// TIA Portal V20 export
// export: Created 2026-08-08T00:00:00.0000000Z, ExportSetting WithDefaults, DisplayName Totally Integrated Automation Portal, DisplayVersion V20, DisplayName TIA Portal Openness, DisplayVersion V20, DisplayName TIA Portal Version Control Interface, DisplayVersion V20, DisplayName STEP 7 Professional, DisplayVersion V20, DisplayName STEP 7 Safety, DisplayVersion V20, DisplayName WinCC Basic/Comfort/Advanced, DisplayVersion V20, DisplayName WinCC Professional, DisplayVersion V20, DisplayName WinCC Unified, DisplayVersion V20
DATA_BLOCK "Valve_Channels_DB"   // DB
{ S7_Optimized_Access := 'TRUE' }
VERSION : 0.1
// Per-valve physical channel assignment table (1..88). All zero until the confirmed valve list / channel schedule is filled in - the mapper and everything downstream treats a zero channel as "use symbolic simulation, no real I/O assigned yet" so this DB is safe to exist unfilled.
// stored: AutoNumber true, IsOnlyStoredInLoadMemory false, IsRetainMemResEnabled false, IsWriteProtectedInAS false, MemoryReserve 100
   VAR
      Channel : Array[1..88] of "UDT_Valve_Config";
   END_VAR
BEGIN
END_DATA_BLOCK
